// TIA Portal V19 export
DATA_BLOCK "Main Control_DB"   // DB1
// stored: InstanceOfName Main Control, InstanceOfType FB
"Main Control"
   // VAR
   //    store : Bool;
   // END_VAR
BEGIN
END_DATA_BLOCK
